(* IEC 61131-3 sources: Elmo_Master/Lasal_PRG/Elmo_EtherCAT_Test_4Axis/Class/TCPIPServer, 1 file *)

(* ---- TCPIPServer.st ---- *)
(*!
<Class
	Name               = "TCPIPServer"
	Revision           = "0.0"
	RealtimeTask       = "false"
	CyclicTask         = "true"
	BackgroundTask     = "false"
	Sigmatek           = "false"
	OSInterface        = "false"
	HighPriority       = "false"
	Automatic          = "false"
	UpdateMode         = "Prescan"
	SharedCommandTable = "true"
	Objectsize         = "(606,120)">
	<Channels>
	</Channels>
	<Network Name="TCPIPServer">
		<!-- List of Components in this network -->
		<Components>
			<Object
				Name       = "_base"
				Class      = "_TCPIPServer"
				Position   = "(218,120)"
				Visualized = "true"
				Remotely   = "true">
				<Channels>
					<Server Name="Control"/>
					<Server Name="ErrorCode"/>
					<Server Name="SemaName01"/>
					<Server Name="SemaName02"/>
					<Server Name="TaskName"/>
					<Client Name="_MultiTask"/>
					<Client Name="_StdLib"/>
					<Client Name="_TaskObjectControl"/>
					<Client Name="Config"/>
					<Client Name="ConnectionsPerRun" Value="1"/>
					<Client Name="MaxConnections" Value="0"/>
					<Client Name="Port"/>
					<Client Name="SigCLib"/>
					<Client Name="SizeOfTXBuffer"/>
					<Client Name="Timeout"/>
				</Channels>
			</Object>
		</Components>
		<Comments>
		</Comments>
		<!-- List of Connections in this network -->
		<Connections>
			<Connection Source="this.Control" Destination="_base.Control" Vertices="(996,210),(824,210),"/>
			<Connection Source="this.ErrorCode" Destination="_base.ErrorCode" Vertices="(996,270),(824,270),"/>
			<Connection Source="this.TaskName" Destination="_base.TaskName" Vertices="(996,330),(824,330),"/>
			<Connection Source="this.SemaName01" Destination="_base.SemaName01" Vertices="(996,390),(824,390),"/>
			<Connection Source="this.SemaName02" Destination="_base.SemaName02" Vertices="(996,450),(824,450),"/>
			<Connection Source="_base.Port" Destination="this.Port" Vertices="(218,210),(38,210),"/>
			<Connection Source="_base.Timeout" Destination="this.Timeout" Vertices="(218,270),(38,270),"/>
			<Connection Source="_base.SizeOfTXBuffer" Destination="this.SizeOfTXBuffer" Vertices="(218,330),(38,330),"/>
			<Connection Source="_base.MaxConnections" Destination="this.MaxConnections" Vertices="(218,390),(38,390),"/>
			<Connection Source="_base.ConnectionsPerRun" Destination="this.ConnectionsPerRun" Vertices="(218,450),(38,450),"/>
			<Connection Source="_base.Config" Destination="this.Config" Vertices="(218,510),(38,510),"/>
			<Connection Source="_base._StdLib" Destination="this._StdLib" Vertices="(218,570),(38,570),"/>
			<Connection Source="_base._MultiTask" Destination="this._MultiTask" Vertices="(218,630),(38,630),"/>
			<Connection Source="_base.SigCLib" Destination="this.SigCLib" Vertices="(218,690),(38,690),"/>
			<Connection Source="_base._TaskObjectControl" Destination="this._TaskObjectControl" Vertices="(218,750),(38,750),"/>
		</Connections>
		<!-- Headerfiles -->
		<Options>
		</Options>
	</Network>
</Class>
*)
#pragma using _TCPIPServer

TCPIPServer : CLASS
: _TCPIPServer
  //Servers:
  //Clients:
  //Variables:
  //Functions:
				//! <Function Comment="Adds a user-class request that moves one connection into the inherited shutdown state." Name="SetSocketParameter"/>
	FUNCTION VIRTUAL GLOBAL SetSocketParameter
		VAR_INPUT
			dSock 	: DINT;
			Cmd 	: DINT;
			SubCmd 	: DINT;
			ParaValue 	: DINT;
		END_VAR
		VAR_OUTPUT
			Retcode 	: DINT;
		END_VAR;
  //Tables:
	FUNCTION @STD
		VAR_OUTPUT
			ret_code	: CONFSTATES;
		END_VAR;
	FUNCTION GLOBAL TAB @CT_;
END_CLASS;

FUNCTION VIRTUAL GLOBAL TCPIPServer::SetSocketParameter
	VAR_INPUT
		dSock 	: DINT;
		Cmd 	: DINT;
		SubCmd 	: DINT;
		ParaValue 	: DINT;
	END_VAR
	VAR_OUTPUT
		Retcode 	: DINT;
	END_VAR
	VAR
		i 	: DINT;
	END_VAR

  // User command 100 requests a controlled disconnect.  Only the inherited
  // FSM state is changed here; _TCPIPServer remains the sole owner of
  // CLOSESOCKET, list removal and the DISCONNECT callback.
  if Cmd = 100 then
    if SubCmd <> 0 then
      Retcode := TCP_SVR_ERR_SET_PARA_INVALID_SUB_CMD;
      RETURN;
    end_if;

    Retcode := TCP_SVR_ERR_INVALID_SOCKET;
    for i := 0 to (MaxConn - 1) do
      if SocketArray[i].dSocket = dSock then
        SocketArray[i].FSM_TCP := _STATE_SHUTDOWN;
        Retcode := TCP_SVR_NO_ERROR;
        exit;
      end_if;
    end_for;
  else
    Retcode := _TCPIPServer::SetSocketParameter(
      dSock:=dSock,
      Cmd:=Cmd,
      SubCmd:=SubCmd,
      ParaValue:=ParaValue
    );
  end_if;

END_FUNCTION
